// SIMATIC STEP 7 (V5.x) project TEMA 5 EJERCICIO 47
// CPU: CPU313 C-2 DP(1)
// station: P_ADR_BUS
// station: Hardware
// station: Equipo SIMATIC 300
// program: Programa S7(1)

SYMBOL_TABLE
"FLANCOS"	DB 1	DB 1
"MANIOBRA"	DB 2	DB 2
"P TICKET"	I 0.0	BOOL
"ENTRADA C FOTOELCTRICA"	I 0.1	BOOL
"P BOTONERA"	I 0.2	BOOL
"SALIDA C FOTOELECTRICA"	I 0.3	BOOL
"CONTADOR"	MW 0	WORD
"Cycle Execution"	OB 1	OB 1
"SUBIR BARRERA ENTRADA"	Q 0.0	BOOL
"BAJAR BARRERA ENTRADA"	Q 0.1	BOOL
"VERDE LIBRE"	Q 0.2	BOOL
"ROJO LLENO"	Q 0.3	BOOL
"SUBIR BARRERA SALIDA"	Q 0.4	BOOL
"BAJAR BARRERA SALIDA"	Q 0.5	BOOL
END_SYMBOL_TABLE

DATA_BLOCK "FLANCOS"	// DB 1
VERSION : 0.1
  STRUCT
   M0 : BOOL ;
   M1 : BOOL ;
   M2 : BOOL ;
   M3 : BOOL ;
   M4 : BOOL ;
   M5 : BOOL ;
   M6 : BOOL ;
   M7 : BOOL ;
   M10 : BOOL ;
   M11 : BOOL ;
   M12 : BOOL ;
   M13 : BOOL ;
   M14 : BOOL ;
   M15 : BOOL ;
   M16 : BOOL ;
   M17 : BOOL ;
   M20 : BOOL ;
   M21 : BOOL ;
   M22 : BOOL ;
   M23 : BOOL ;
   M24 : BOOL ;
   M25 : BOOL ;
   M26 : BOOL ;
   M27 : BOOL ;
  END_STRUCT ;	
BEGIN
END_DATA_BLOCK

DATA_BLOCK "MANIOBRA"	// DB 2
VERSION : 0.1
  STRUCT
   MO : BOOL ;
   M1 : BOOL ;
   M2 : BOOL ;
   M3 : BOOL ;
   M4 : BOOL ;
   M5 : BOOL ;
   M6 : BOOL ;
   M7 : BOOL ;
   M10 : BOOL ;
   M11 : BOOL ;
   M12 : BOOL ;
   M13 : BOOL ;
   M14 : BOOL ;
   M15 : BOOL ;
   M16 : BOOL ;
   M17 : BOOL ;
  END_STRUCT ;	
BEGIN
END_DATA_BLOCK

ORGANIZATION_BLOCK "Cycle Execution"	// OB 1
TITLE = "Main Program Sweep (Cycle)"
//PARKING.
//
VERSION : 0.1
VAR_TEMP
  OB1_EV_CLASS : BYTE ;	//Bits 0-3 = 1 (Coming event), Bits 4-7 = 1 (Event class 1)
  OB1_SCAN_1 : BYTE ;	//1 (Cold restart scan 1 of OB 1), 3 (Scan 2-n of OB 1)
  OB1_PRIORITY : BYTE ;	//Priority of OB Execution
  OB1_OB_NUMBR : BYTE ;	//1 (Organization block 1, OB1)
  OB1_RESERVED_1 : BYTE ;	//Reserved for system
  OB1_RESERVED_2 : BYTE ;	//Reserved for system
  OB1_PREV_CYCLE : INT ;	//Cycle time of previous OB1 scan (milliseconds)
  OB1_MIN_CYCLE : INT ;	//Minimum cycle time of OB1 (milliseconds)
  OB1_MAX_CYCLE : INT ;	//Maximum cycle time of OB1 (milliseconds)
  OB1_DATE_TIME : DATE_AND_TIME ;	//Date and time OB1 started
END_VAR
BEGIN
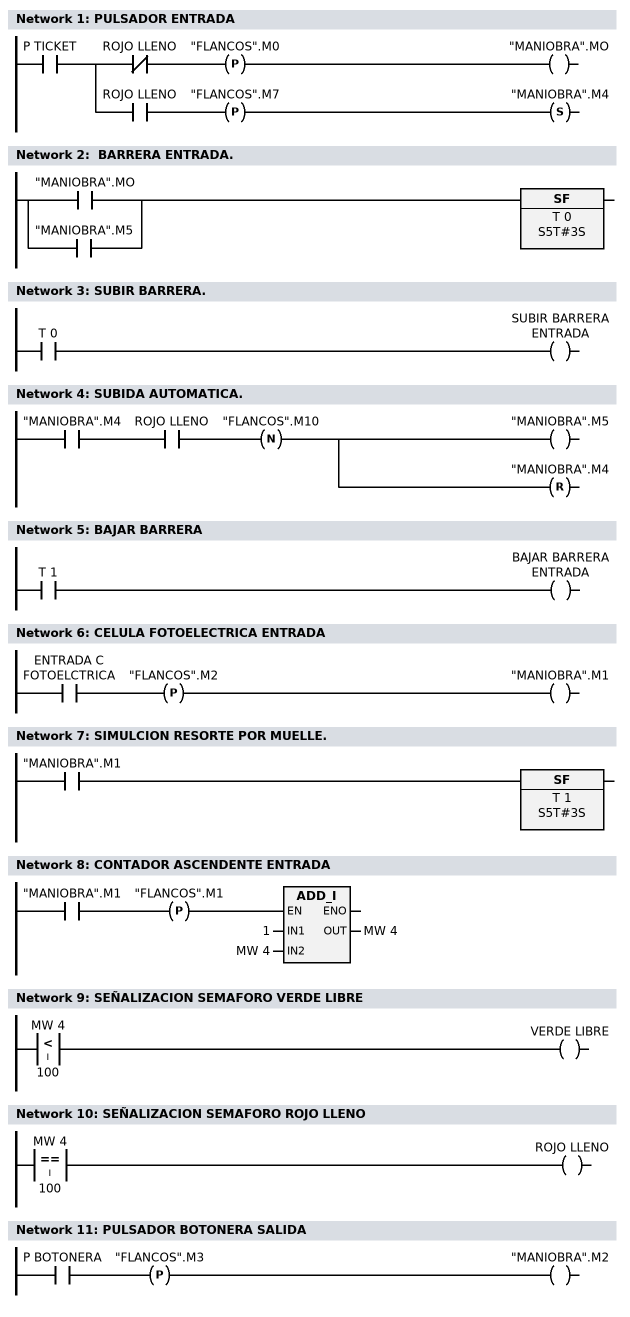
NETWORK
TITLE = PULSADOR ENTRADA
//ENPENDERA UN TICKET (SIMBOLICO CARECE DE IMPORTANCIA EN EL PROGRAMA).
//LEVANTARA LA BARRERA.
//MANIOBRA 4 SE ENCARGA DE REGISTRAR EL PULSO CUANDO ESTA LLENO Y PREPARAR EL 
//PROGRAMA QUE EJECUTARA LA SUBIDA DE BARRERA AUTOMATICA CUANDO QUEDA UNA PLAZA 
//LIBRE.
      A     "P TICKET";
      =     L 20.0;
      A     L 20.0;
      AN    "ROJO LLENO";
      FP    "FLANCOS".M0;
      =     "MANIOBRA".MO;
      A     L 20.0;
      A     "ROJO LLENO";
      FP    "FLANCOS".M7;
      S     "MANIOBRA".M4;
NETWORK
TITLE =  BARRERA ENTRADA.
//PARA SIMULAR EL PISTON UTILIZO UN TEMPORIZADOR A LA DESCONEXION QUE MANTENDRA 
//ALIMENTADA UNA SALIDA DURANE 3SEG. QUE EL TIEMPO QUE TARDA LA BARRERA EN HACER 
//SU RECORRIDO
      O     "MANIOBRA".MO;
      O     "MANIOBRA".M5;
      L     S5T#3S;
      SF    T 0;
NETWORK
TITLE = SUBIR BARRERA.
      A     T 0;
      =     "SUBIR BARRERA ENTRADA";
NETWORK
TITLE = SUBIDA AUTOMATICA.
//SE PRODUCE CUANDO EL PARKING ESTA LLENO Y UN USUARIO PULSA EL 
//P.ENTRADA.AUTOMATICAMENTE SE  SUBIRA CUANDO SALGA UN COCHE. 
      A     "MANIOBRA".M4;
      A     "ROJO LLENO";
      FN    "FLANCOS".M10;
      =     "MANIOBRA".M5;
      R     "MANIOBRA".M4;
NETWORK
TITLE = BAJAR BARRERA 
      A     T 1;
      =     "BAJAR BARRERA ENTRADA";
NETWORK
TITLE = CELULA FOTOELECTRICA ENTRADA
//BAJA BARRERA Y SUMA UNO A CONTADOR.
      A     "ENTRADA C FOTOELCTRICA";
      FP    "FLANCOS".M2;
      =     "MANIOBRA".M1;
NETWORK
TITLE = SIMULCION RESORTE POR MUELLE.
//EL FUNCIONAMIENTO ES EL MISMO QUE EN EL CASO ANTERIOR.
      A     "MANIOBRA".M1;
      L     S5T#3S;
      SF    T 1;
NETWORK
TITLE = CONTADOR ASCENDENTE ENTRADA
      A     "MANIOBRA".M1;
      FP    "FLANCOS".M1;
      JNB   _001;
      L     1;
      L     MW 4;
      +I;
      T     MW 4;
_001: NOP   0;
NETWORK
TITLE = SEÑALIZACION SEMAFORO VERDE LIBRE
//ESTARA ENCENDIDA SIEMPRE QUE LA CANTIDAD DE COCHES SEA INFERIOR A 100.
      L     MW 4;
      L     100;
      <I;
      =     "VERDE LIBRE";
NETWORK
TITLE = SEÑALIZACION SEMAFORO ROJO LLENO
//SE ENCENDERA CUANDO LA CANTIDAD DE COCHESS SEA IGUAL A 100 Y NO PERMITIRA LA 
//ENTRADA HASTA QUE SALGA 1.
      L     MW 4;
      L     100;
      ==I;
      =     "ROJO LLENO";
NETWORK
TITLE = PULSADOR BOTONERA SALIDA
      A     "P BOTONERA";
      FP    "FLANCOS".M3;
      =     "MANIOBRA".M2;
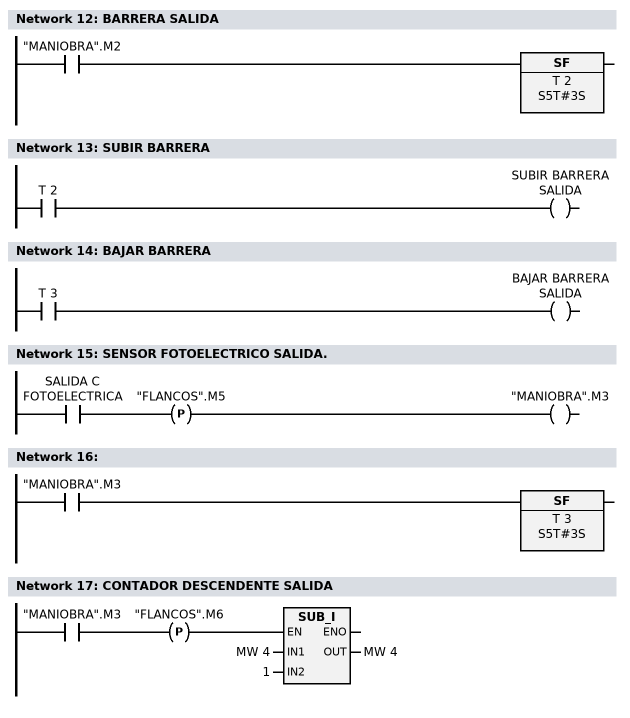
NETWORK
TITLE = BARRERA SALIDA
      A     "MANIOBRA".M2;
      L     S5T#3S;
      SF    T 2;
NETWORK
TITLE = SUBIR BARRERA
      A     T 2;
      =     "SUBIR BARRERA SALIDA";
NETWORK
TITLE = BAJAR BARRERA
      A     T 3;
      =     "BAJAR BARRERA SALIDA";
NETWORK
TITLE = SENSOR FOTOELECTRICO SALIDA.
//BAJA LA BARRERA Y RESTA UNO EN EL CONTADOR.
      A     "SALIDA C FOTOELECTRICA";
      FP    "FLANCOS".M5;
      =     "MANIOBRA".M3;
NETWORK
TITLE =
      A     "MANIOBRA".M3;
      L     S5T#3S;
      SF    T 3;
NETWORK
TITLE = CONTADOR DESCENDENTE SALIDA
      A     "MANIOBRA".M3;
      FP    "FLANCOS".M6;
      JNB   _002;
      L     MW 4;
      L     1;
      -I;
      T     MW 4;
_002: NOP   0;
END_ORGANIZATION_BLOCK
